// Mitsubishi GX Works2 project: k04   PLC: Q02/Q02H

PROGRAM MAIN
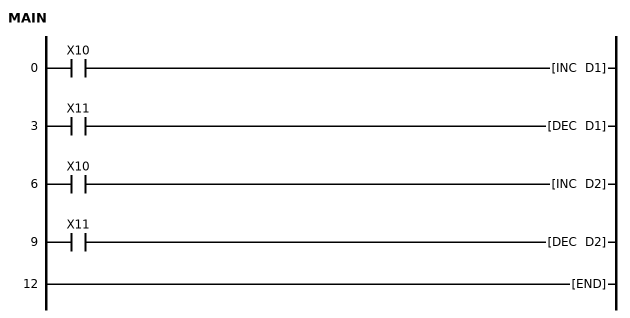
0     LD      X10
      INC     D1
3     LD      X11
      DEC     D1
6     LD      X10
      INC     D2
9     LD      X11
      DEC     D2
12    END
END_PROGRAM
